Staubli VAL3: ack.pgx

public program ack(num x_nHeaderTime, num x_nElapsedTime)
begin

  // display time between valid trajectory point received and ACK sent

  userPageSet("uxMonitor", "lblHeaderTime", "innerHTML", toString(".4", x_nHeaderTime))
  userPageSet("uxMonitor", "lblElapsedTime", "innerHTML", toString(".4", x_nElapsedTime))

end
